TYPE ST_Curtain_op :
STRUCT
	Open	 AT%Q* : BOOL;
	Close	 AT%Q* : BOOL;	
END_STRUCT
END_TYPE

(* stored: Version 1.1.0.1, ProductVersion 3.1.4024.12
   DUT ST_Curtain_op: Id {01eab23d-270b-4dd1-ad77-79ea239e143d} *)
